TYPE T_HEART_BEAT : UDINT; END_TYPE		// Signal used to check the heart beat (over ADS)

(* stored: Version 1.1.0.1, ProductVersion 3.1.4026.18
   DUT T_HEART_BEAT: Id {fe88bdee-e9ac-4067-b8f5-90cd09fd91cc} *)
